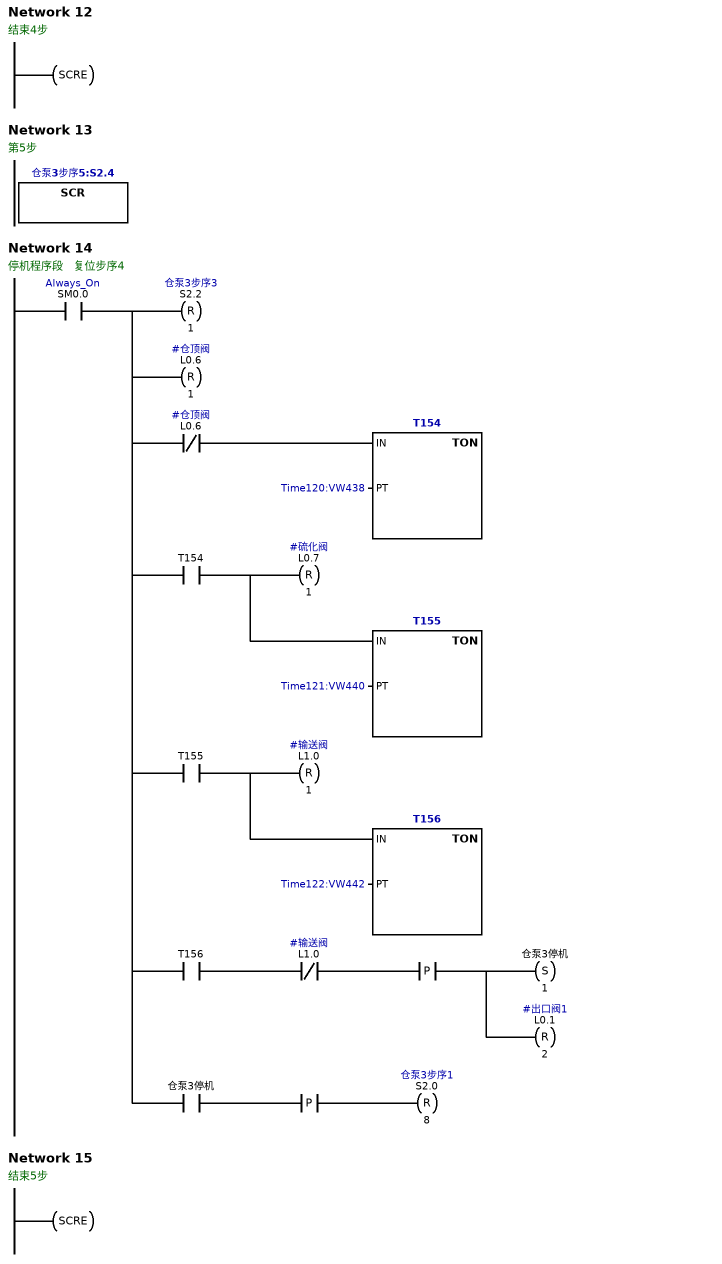
[picture p48: SBR18 networks 12-15]
Network 12
// 结束4步
SCRE
Network 13
// 第5步 
LSCR   仓泵3步序5:S2.4
Network 14
// 停机程序段   复位步序4 
// (network saved uncompiled; LAD cells follow)
// row 0: c0 -| |- Always_On:SM0.0 v  c1 -(R) 仓泵3步序3:S2.2, 1
// row 1: c0 ^v  c1 -(R) #仓顶阀:L0.6, 1
// row 2: c0 ^v  c1 -|/|- #仓顶阀:L0.6  c2 --  c3 [TON T154 IN:=power@row2, PT:=Time120:VW438]
// row 3: c0 ^v  c3 [box]
// row 4: c0 ^v  c1 -| |- T154 v  c2 -(R) #硫化阀:L0.7, 1
// row 5: c0 ^v  c1 ^  c2 --  c3 [TON T155 IN:=power@row5, PT:=Time121:VW440]
// row 6: c0 ^v  c3 [box]
// row 7: c0 ^v  c1 -| |- T155 v  c2 -(R) #输送阀:L1.0, 1
// row 8: c0 ^v  c1 ^  c2 --  c3 [TON T156 IN:=power@row8, PT:=Time122:VW442]
// row 9: c0 ^v  c3 [box]
// row 10: c0 ^v  c1 -| |- T156  c2 -|/|- #输送阀:L1.0  c3 -|P|-  v  c4 -(S) 仓泵3停机, 1
// row 11: c0 ^v  c3 ^  c4 -(R) #出口阀1:L0.1, 2
// row 12: c0 ^  c1 -| |- 仓泵3停机  c2 -|P|-  c3 -(R) 仓泵3步序1:S2.0, 8
Network 15
// 结束5步
SCRE
END_SUBROUTINE_BLOCK

SUBROUTINE_BLOCK 除尘器下料1:SBR19
TITLE=除尘器下料程序子程序说明   ：该子程序可用于除尘器下料程序  调用该子程序只需要填好子程序接口参数   然后核对子程序内部计数器有没有重复使用  有重复更改计数器  没有重复填好接口参数可直接使用
// 
// 从上往下依次的子程序接口
// 
// 使能
//  除尘器下料许可
// 系统错误
// 除尘器下料上下阀门自动位
// 除尘器下料阀上部Q点
// 除尘器下料阀下部Q点
// 除尘器气锤自动位
// 除尘器气碟自动位
// 除尘器中转气锤自动位
// 除尘器中转气碟自动位
// 上部阀门设定次数
// 下部阀门设定次数
// 上部阀门显示次数
// 下部阀门显示次数
VAR_INPUT
Sure:BOOL;	// L0.0 除尘器下料许可
END_VAR
VAR_IN_OUT
Error:BOOL;	// L0.1 系统错误
除尘器下料阀:BOOL;	// L0.2 除尘器下料阀ZD位 驱动两个阀门上下交替运行
除尘器下料阀上部:BOOL;	// L0.3 下料阀的上部阀门
除尘器下料阀下部:BOOL;	// L0.4 下料阀的下部阀门
除尘器气锤:BOOL;	// L0.5 气锤
除尘器气碟:BOOL;	// L0.6 气碟
除尘器中转气锤:BOOL;	// L0.7 中转气锤
除尘器中转气碟:BOOL;	// L1.0 中转气碟
上部次数设定:INT;	// LW2 上部阀运行次数设定
下部次数设定:INT;	// LW4 下部阀运行次数设定
上部次数显示:INT;	// LW6 上部阀运行次数显示
下部次数显示:INT;	// LW8 下部阀运行次数显示
END_VAR
BEGIN
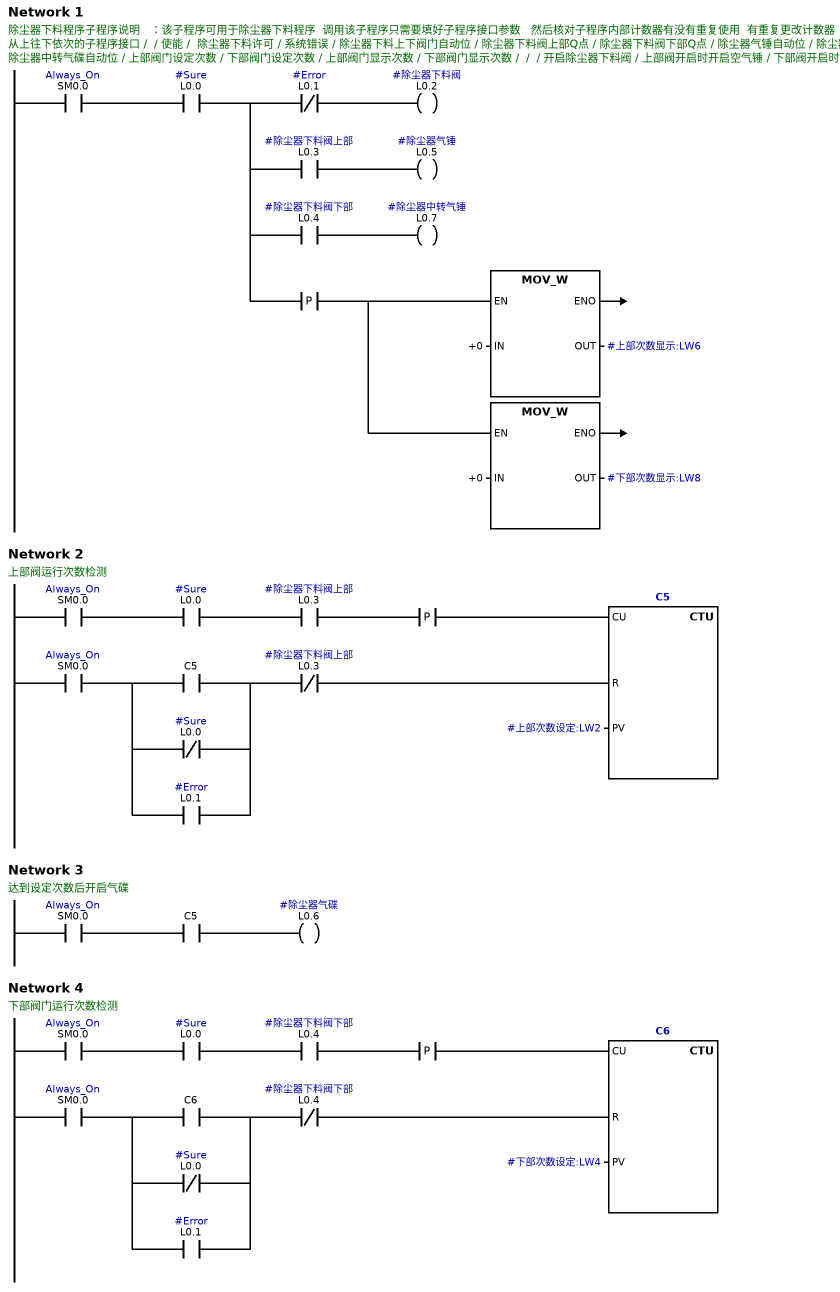
Network 1
// 除尘器下料程序子程序说明   ：该子程序可用于除尘器下料程序  调用该子程序只需要填好子程序接口参数   然后核对子程序内部计数器有没有重复使用  有重复更改计数器  没有重复填好接口参数可直接使用
// 
// 从上往下依次的子程序接口
// 
// 使能
//  除尘器下料许可
// 系统错误
// 除尘器下料上下阀门自动位
// 除尘器下料阀上部Q点
// 除尘器下料阀下部Q点
// 除尘器气锤自动位
// 除尘器气碟自动位
// 除尘器中转气锤自动位
// 除尘器中转气碟自动位
// 上部阀门设定次数
// 下部阀门设定次数
// 上部阀门显示次数
// 下部阀门显示次数
// 
// 
// 开启除尘器下料阀
// 上部阀开启时开启空气锤
// 下部阀开启时开启中转空气锤1
// 上部阀开启设定次数后开启气碟
// 下部阀开启设定次数后开启中转
LD     Always_On:SM0.0
A      #Sure:L0.0
LPS
AN     #Error:L0.1
=      #除尘器下料阀:L0.2
LRD
A      #除尘器下料阀上部:L0.3
=      #除尘器气锤:L0.5
LRD
A      #除尘器下料阀下部:L0.4
=      #除尘器中转气锤:L0.7
LPP
EU
MOVW   +0, #上部次数显示:LW6
MOVW   +0, #下部次数显示:LW8
Network 2
// 上部阀运行次数检测
LD     Always_On:SM0.0
A      #Sure:L0.0
A      #除尘器下料阀上部:L0.3
EU
LD     Always_On:SM0.0
LD     C5
ON     #Sure:L0.0
O      #Error:L0.1
ALD
AN     #除尘器下料阀上部:L0.3
CTU    C5, #上部次数设定:LW2
Network 3
// 达到设定次数后开启气碟
LD     Always_On:SM0.0
A      C5
=      #除尘器气碟:L0.6
Network 4
// 下部阀门运行次数检测
LD     Always_On:SM0.0
A      #Sure:L0.0
A      #除尘器下料阀下部:L0.4
EU
LD     Always_On:SM0.0
LD     C6
ON     #Sure:L0.0
O      #Error:L0.1
ALD
AN     #除尘器下料阀下部:L0.4
CTU    C6, #下部次数设定:LW4
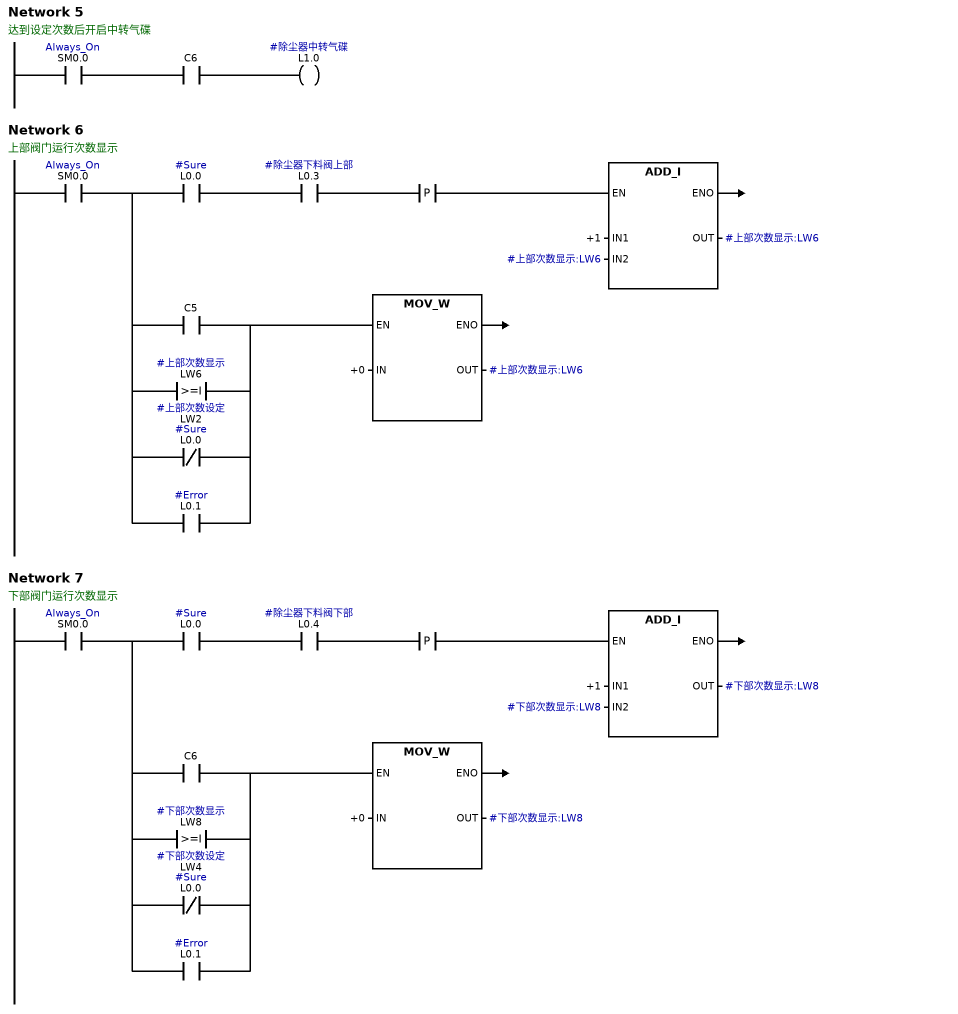
Network 5
// 达到设定次数后开启中转气碟
LD     Always_On:SM0.0
A      C6
=      #除尘器中转气碟:L1.0
Network 6
// 上部阀门运行次数显示
LD     Always_On:SM0.0
LPS
A      #Sure:L0.0
A      #除尘器下料阀上部:L0.3
EU
+I     +1, #上部次数显示:LW6
LPP
LD     C5
OW>=   #上部次数显示:LW6, #上部次数设定:LW2
ON     #Sure:L0.0
O      #Error:L0.1
ALD
MOVW   +0, #上部次数显示:LW6
Network 7
// 下部阀门运行次数显示
LD     Always_On:SM0.0
LPS
A      #Sure:L0.0
A      #除尘器下料阀下部:L0.4
EU
+I     +1, #下部次数显示:LW8
LPP
LD     C6
OW>=   #下部次数显示:LW8, #下部次数设定:LW4
ON     #Sure:L0.0
O      #Error:L0.1
ALD
MOVW   +0, #下部次数显示:LW8
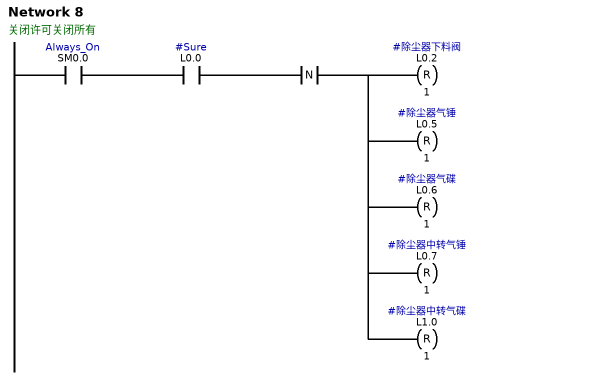
Network 8
// 关闭许可关闭所有
LD     Always_On:SM0.0
A      #Sure:L0.0
ED
R      #除尘器下料阀:L0.2, 1
R      #除尘器气锤:L0.5, 1
R      #除尘器气碟:L0.6, 1
R      #除尘器中转气锤:L0.7, 1
R      #除尘器中转气碟:L1.0, 1
END_SUBROUTINE_BLOCK

SUBROUTINE_BLOCK PauseUpValve5Group:SBR20
TITLE=
VAR_IN_OUT
Hand:BOOL;	// L0.0 手动信号
Auto:BOOL;	// L0.1 自动信号
Err:BOOL;	// L0.2 系统故障
UpValve1:BOOL;	// L0.3 提升阀1
UpValve2:BOOL;	// L0.4 提升阀2
UpValve3:BOOL;	// L0.5 提升阀3
UpValve4:BOOL;	// L0.6 提升阀4
UpValve5:BOOL;	// L0.7 提升阀5
Pulse1:BOOL;	// L1.0 脉冲阀1
Pulse2:BOOL;	// L1.1 脉冲阀2
Pulse3:BOOL;	// L1.2 脉冲阀3
Pulse4:BOOL;	// L1.3 脉冲阀4
Pulse5:BOOL;	// L1.4 脉冲阀5
UpValveRuntime:INT;	// LW2 提举阀运行时间
UpValveStoptime:INT;	// LW4 提举阀停止时间
PulseRuntime:INT;	// LW6 脉冲阀运行时间
PulseStoptime:INT;	// LW8 脉冲阀停止时间
END_VAR
BEGIN
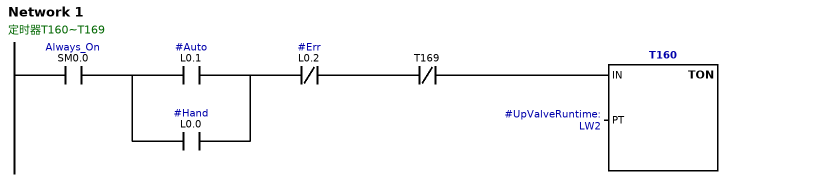
Network 1
// 定时器T160~T169
LD     Always_On:SM0.0
LD     #Auto:L0.1
O      #Hand:L0.0
ALD
AN     #Err:L0.2
AN     T169
TON    T160, #UpValveRuntime:LW2
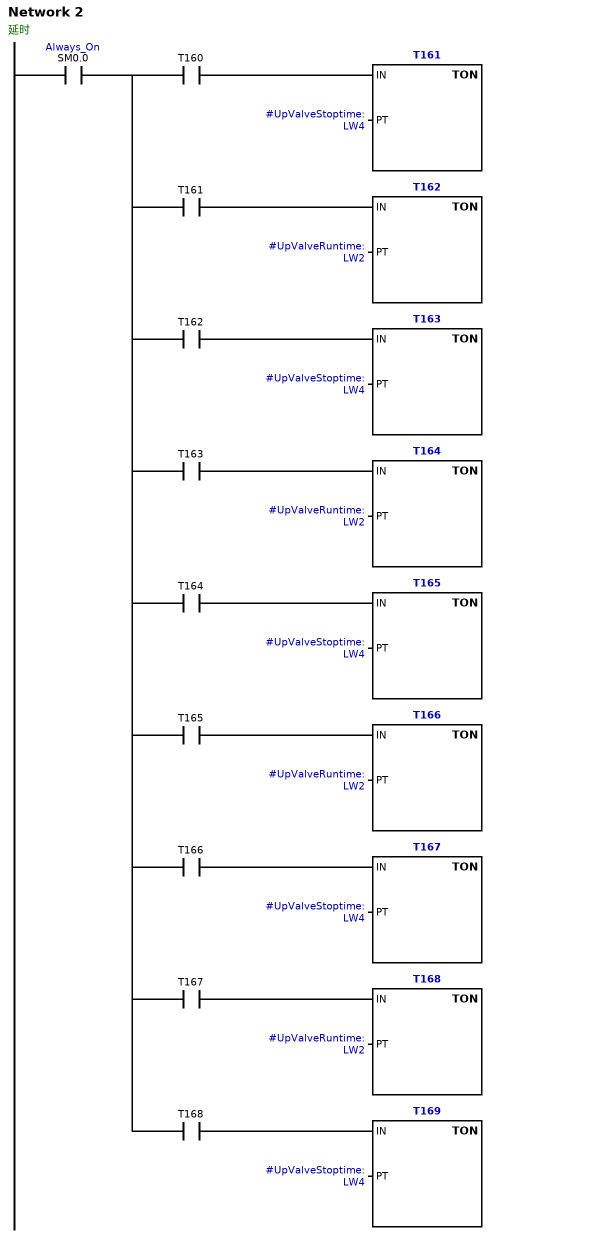
Network 2
// 延时
LD     Always_On:SM0.0
LPS
A      T160
TON    T161, #UpValveStoptime:LW4
LRD
A      T161
TON    T162, #UpValveRuntime:LW2
LRD
A      T162
TON    T163, #UpValveStoptime:LW4
LRD
A      T163
TON    T164, #UpValveRuntime:LW2
LRD
A      T164
TON    T165, #UpValveStoptime:LW4
LRD
A      T165
TON    T166, #UpValveRuntime:LW2
LRD
A      T166
TON    T167, #UpValveStoptime:LW4
LRD
A      T167
TON    T168, #UpValveRuntime:LW2
LPP
A      T168
TON    T169, #UpValveStoptime:LW4
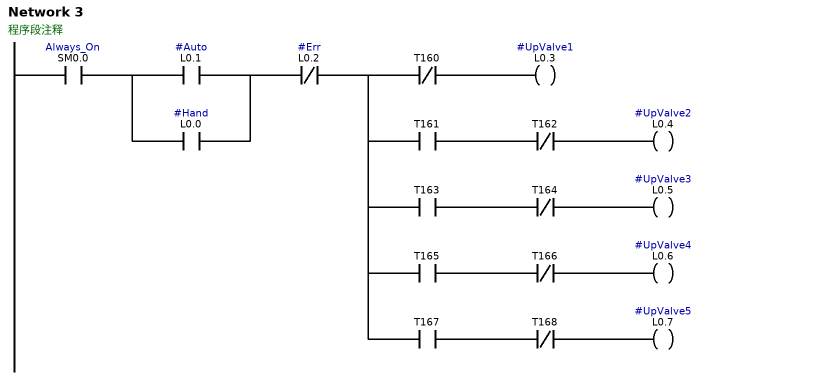
Network 3
//  程序段注释
LD     Always_On:SM0.0
LD     #Auto:L0.1
O      #Hand:L0.0
ALD
AN     #Err:L0.2
LPS
AN     T160
=      #UpValve1:L0.3
LRD
A      T161
AN     T162
=      #UpValve2:L0.4
LRD
A      T163
AN     T164
=      #UpValve3:L0.5
LRD
A      T165
AN     T166
=      #UpValve4:L0.6
LPP
A      T167
AN     T168
=      #UpValve5:L0.7
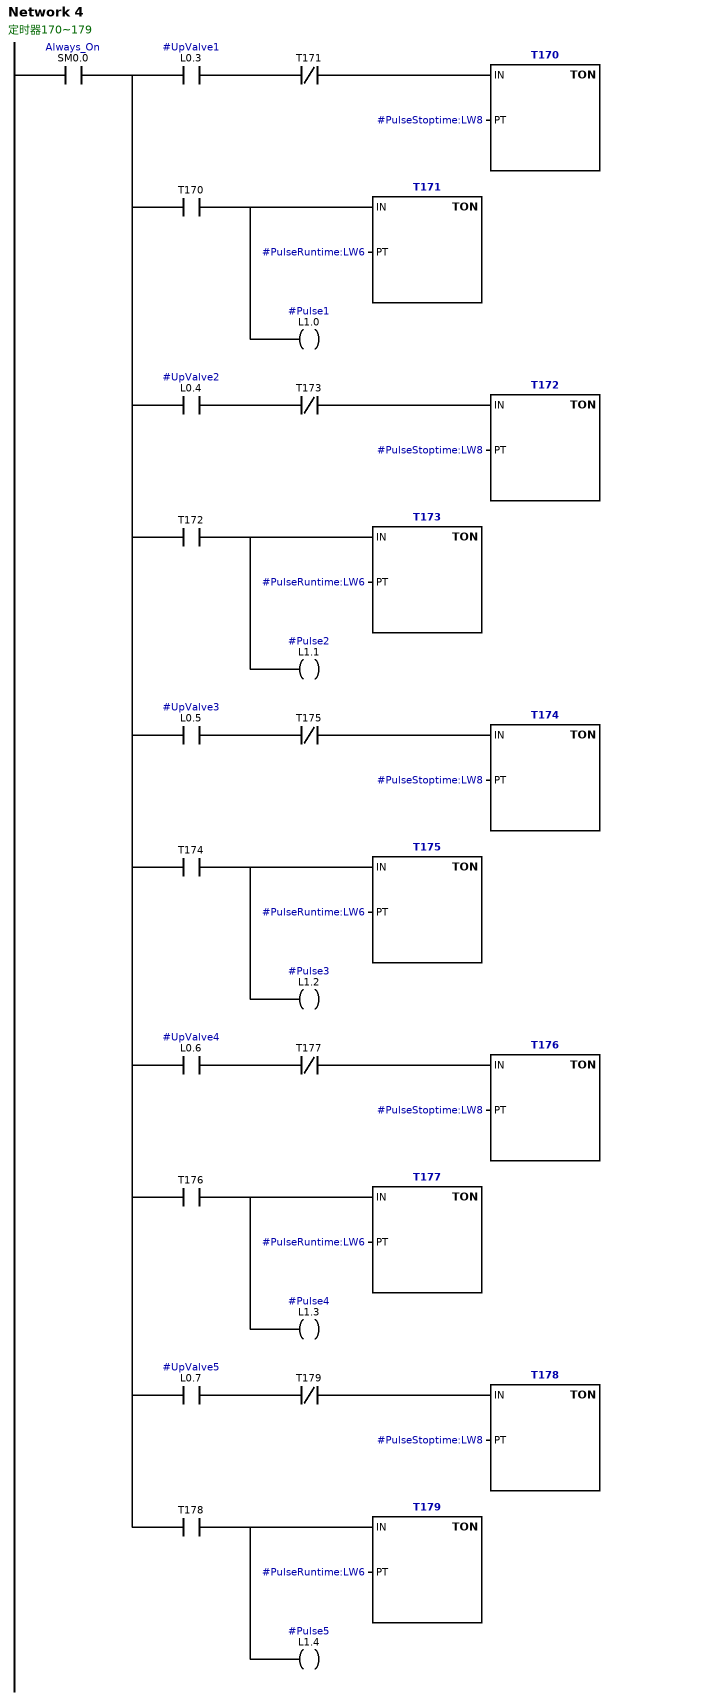
Network 4
// 定时器170~179
LD     Always_On:SM0.0
LPS
A      #UpValve1:L0.3
AN     T171
TON    T170, #PulseStoptime:LW8
LRD
A      T170
TON    T171, #PulseRuntime:LW6
=      #Pulse1:L1.0
LRD
A      #UpValve2:L0.4
AN     T173
TON    T172, #PulseStoptime:LW8
LRD
A      T172
TON    T173, #PulseRuntime:LW6
=      #Pulse2:L1.1
LRD
A      #UpValve3:L0.5
AN     T175
TON    T174, #PulseStoptime:LW8
LRD
A      T174
TON    T175, #PulseRuntime:LW6
=      #Pulse3:L1.2
LRD
A      #UpValve4:L0.6
AN     T177
TON    T176, #PulseStoptime:LW8
LRD
A      T176
TON    T177, #PulseRuntime:LW6
=      #Pulse4:L1.3
LRD
A      #UpValve5:L0.7
AN     T179
TON    T178, #PulseStoptime:LW8
LPP
A      T178
TON    T179, #PulseRuntime:LW6
=      #Pulse5:L1.4
END_SUBROUTINE_BLOCK

SUBROUTINE_BLOCK 双除尘器切换1:SBR21
TITLE=
VAR_INPUT
IN_T1:BOOL;	// L0.0 
IN_T2:BOOL;	// L0.1 
END_VAR
VAR_IN_OUT
进口阀1:BOOL;	// L0.2 
出口阀1:BOOL;	// L0.3 
脉冲仪1:BOOL;	// L0.4 
进口阀2:BOOL;	// L0.5 
出口阀2:BOOL;	// L0.6 
脉冲仪2:BOOL;	// L0.7 
引风机1:BOOL;	// L1.0 
引风机2:BOOL;	// L1.1 
State1:BOOL;	// L1.2 除尘器1 切换中
State2:BOOL;	// L1.3 除尘器2 切换中
END_VAR
BEGIN
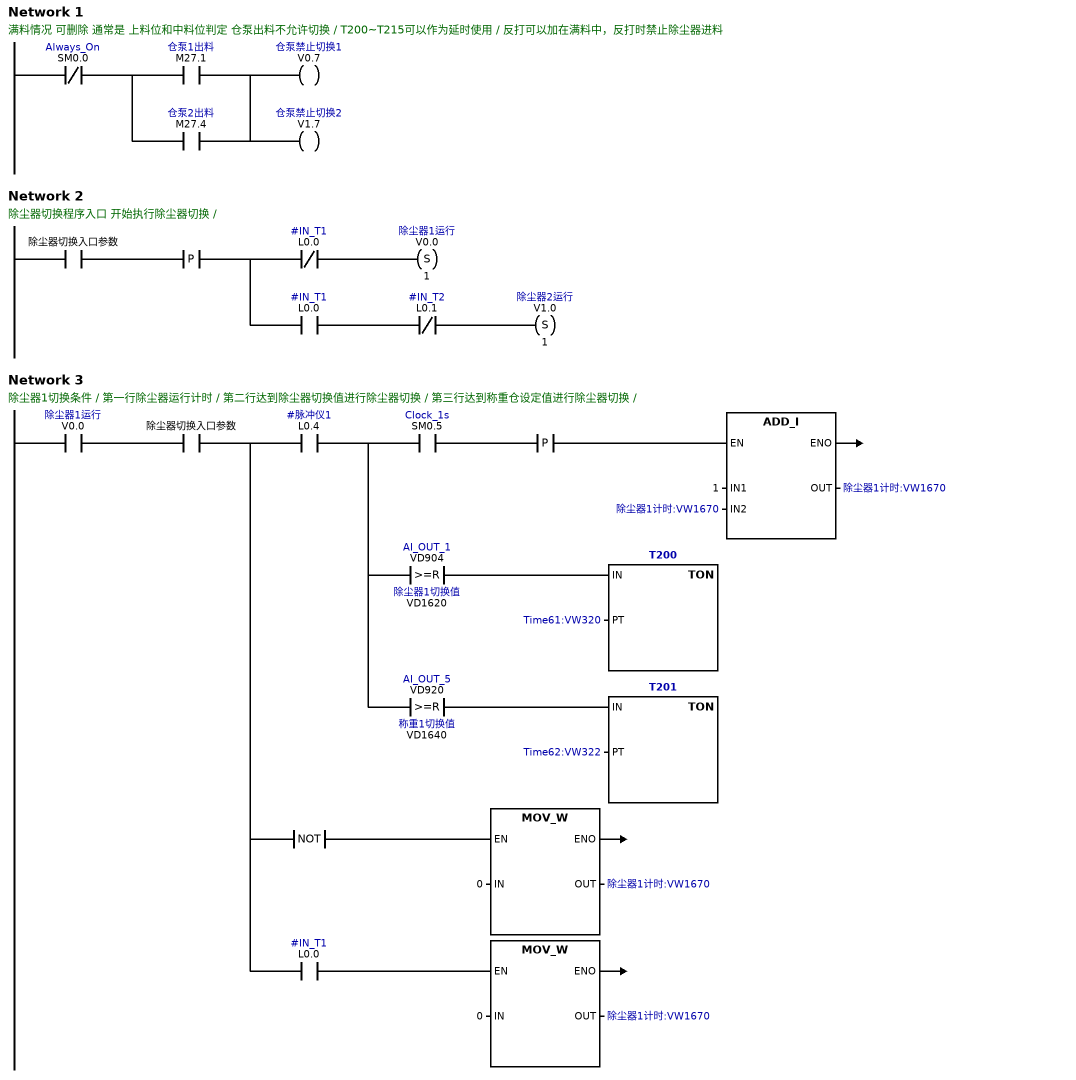
Network 1
// 满料情况 可删除 通常是 上料位和中料位判定 仓泵出料不允许切换
// T200~T215可以作为延时使用
// 反打可以加在满料中，反打时禁止除尘器进料
LDN    Always_On:SM0.0
LD     仓泵1出料:M27.1
O      仓泵2出料:M27.4
ALD
=      仓泵禁止切换1:V0.7
=      仓泵禁止切换2:V1.7
Network 2
//  除尘器切换程序入口 开始执行除尘器切换
// 
// (network saved uncompiled; LAD cells follow)
// row 0: c0 -| |- 除尘器切换入口参数  c1 -|P|-  v  c2 -|/|- #IN_T1:L0.0  c3 -(S) 除尘器1运行:V0.0, 1
// row 1: c1 ^  c2 -| |- #IN_T1:L0.0  c3 -|/|- #IN_T2:L0.1  c4 -(S) 除尘器2运行:V1.0, 1
Network 3
// 除尘器1切换条件
// 第一行除尘器运行计时
// 第二行达到除尘器切换值进行除尘器切换
// 第三行达到称重仓设定值进行除尘器切换
// 
// (network saved uncompiled; LAD cells follow)
// row 0: c0 -| |- 除尘器1运行:V0.0  c1 -| |- 除尘器切换入口参数 v  c2 -| |- #脉冲仪1:L0.4 v  c3 -| |- Clock_1s:SM0.5  c4 -|P|-  c5 --  c6 [ADD_I EN:=power@row0, IN1:=1, IN2:=除尘器1计时:VW1670, ENO=>power, OUT=>除尘器1计时:VW1670]  c7 ->
// row 1: c1 ^v  c2 ^v  c6 [box]
// row 2: c1 ^v  c2 ^v  c3 -|>=R|- AI_OUT_1:VD904, 除尘器1切换值:VD1620  c4 --  c5 [TON T200 IN:=power@row2, PT:=Time61:VW320]
// row 3: c1 ^v  c2 ^v  c5 [box]
// row 4: c1 ^v  c2 ^  c3 -|>=R|- AI_OUT_5:VD920, 称重1切换值:VD1640  c4 --  c5 [TON T201 IN:=power@row4, PT:=Time62:VW322]
// row 5: c1 ^v  c5 [box]
// row 6: c1 ^v  c2 -|NOT|-  c3 --  c4 [MOV_W EN:=power@row6, IN:=0, ENO=>power, OUT=>除尘器1计时:VW1670]  c5 ->
// row 7: c1 ^v  c4 [box]
// row 8: c1 ^  c2 -| |- #IN_T1:L0.0  c3 --  c4 [MOV_W EN:=power@row8, IN:=0, ENO=>power, OUT=>除尘器1计时:VW1670]  c5 ->
// row 9: c4 [box]
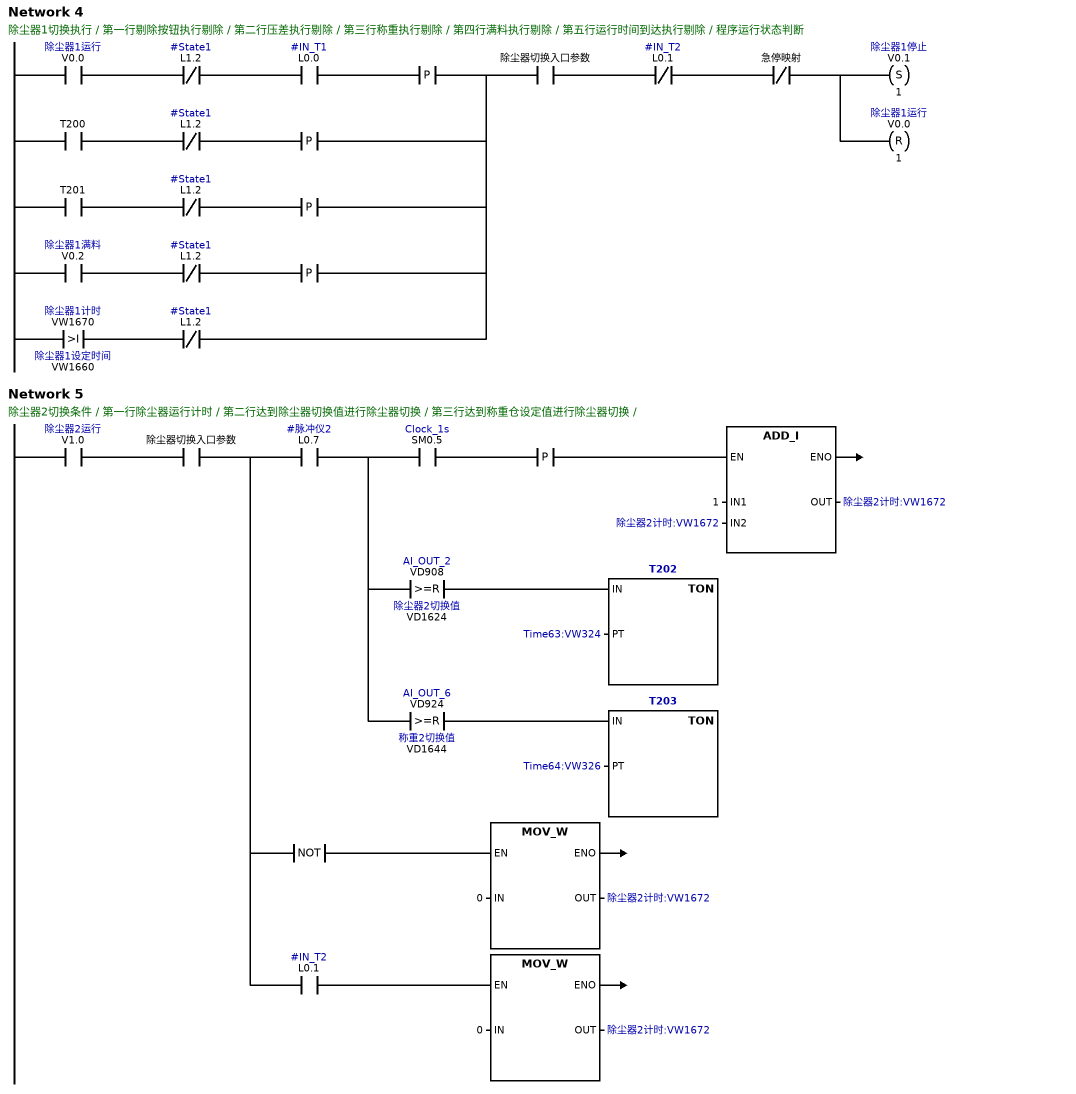
Network 4
// 除尘器1切换执行
// 第一行剔除按钮执行剔除
// 第二行压差执行剔除
// 第三行称重执行剔除
// 第四行满料执行剔除
// 第五行运行时间到达执行剔除
// 程序运行状态判断
// (network saved uncompiled; LAD cells follow)
// row 0: c0 -| |- 除尘器1运行:V0.0  c1 -|/|- #State1:L1.2  c2 -| |- #IN_T1:L0.0  c3 -|P|-  v  c4 -| |- 除尘器切换入口参数  c5 -|/|- #IN_T2:L0.1  c6 -|/|- 急停映射 v  c7 -(S) 除尘器1停止:V0.1, 1
// row 1: c0 -| |- T200  c1 -|/|- #State1:L1.2  c2 -|P|-  c3 -- ^v  c6 ^  c7 -(R) 除尘器1运行:V0.0, 1
// row 2: c0 -| |- T201  c1 -|/|- #State1:L1.2  c2 -|P|-  c3 -- ^v
// row 3: c0 -| |- 除尘器1满料:V0.2  c1 -|/|- #State1:L1.2  c2 -|P|-  c3 -- ^v
// row 4: c0 -|>I|- 除尘器1计时:VW1670, 除尘器1设定时间:VW1660  c1 -|/|- #State1:L1.2  c2 --  c3 -- ^
Network 5
// 除尘器2切换条件
// 第一行除尘器运行计时
// 第二行达到除尘器切换值进行除尘器切换
// 第三行达到称重仓设定值进行除尘器切换
// 
// (network saved uncompiled; LAD cells follow)
// row 0: c0 -| |- 除尘器2运行:V1.0  c1 -| |- 除尘器切换入口参数 v  c2 -| |- #脉冲仪2:L0.7 v  c3 -| |- Clock_1s:SM0.5  c4 -|P|-  c5 --  c6 [ADD_I EN:=power@row0, IN1:=1, IN2:=除尘器2计时:VW1672, ENO=>power, OUT=>除尘器2计时:VW1672]  c7 ->
// row 1: c1 ^v  c2 ^v  c6 [box]
// row 2: c1 ^v  c2 ^v  c3 -|>=R|- AI_OUT_2:VD908, 除尘器2切换值:VD1624  c4 --  c5 [TON T202 IN:=power@row2, PT:=Time63:VW324]
// row 3: c1 ^v  c2 ^v  c5 [box]
// row 4: c1 ^v  c2 ^  c3 -|>=R|- AI_OUT_6:VD924, 称重2切换值:VD1644  c4 --  c5 [TON T203 IN:=power@row4, PT:=Time64:VW326]
// row 5: c1 ^v  c5 [box]
// row 6: c1 ^v  c2 -|NOT|-  c3 --  c4 [MOV_W EN:=power@row6, IN:=0, ENO=>power, OUT=>除尘器2计时:VW1672]  c5 ->
// row 7: c1 ^v  c4 [box]
// row 8: c1 ^  c2 -| |- #IN_T2:L0.1  c3 --  c4 [MOV_W EN:=power@row8, IN:=0, ENO=>power, OUT=>除尘器2计时:VW1672]  c5 ->
// row 9: c4 [box]
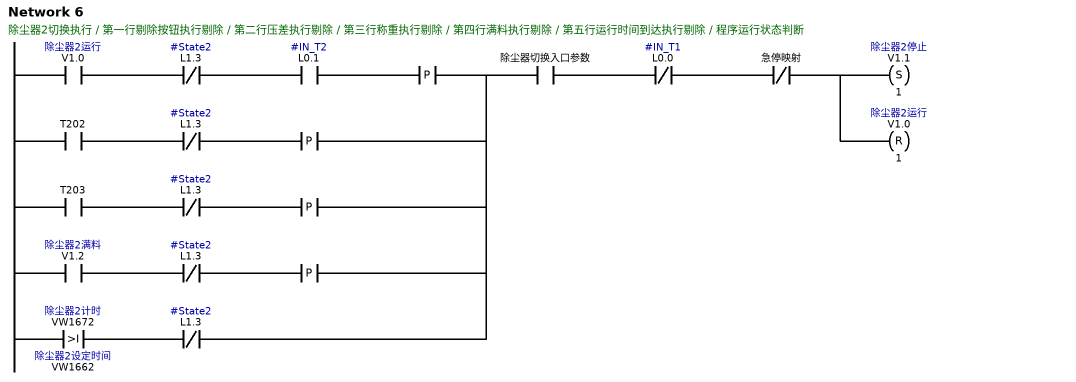
Network 6
// 除尘器2切换执行
// 第一行剔除按钮执行剔除
// 第二行压差执行剔除
// 第三行称重执行剔除
// 第四行满料执行剔除
// 第五行运行时间到达执行剔除
// 程序运行状态判断
// (network saved uncompiled; LAD cells follow)
// row 0: c0 -| |- 除尘器2运行:V1.0  c1 -|/|- #State2:L1.3  c2 -| |- #IN_T2:L0.1  c3 -|P|-  v  c4 -| |- 除尘器切换入口参数  c5 -|/|- #IN_T1:L0.0  c6 -|/|- 急停映射 v  c7 -(S) 除尘器2停止:V1.1, 1
// row 1: c0 -| |- T202  c1 -|/|- #State2:L1.3  c2 -|P|-  c3 -- ^v  c6 ^  c7 -(R) 除尘器2运行:V1.0, 1
// row 2: c0 -| |- T203  c1 -|/|- #State2:L1.3  c2 -|P|-  c3 -- ^v
// row 3: c0 -| |- 除尘器2满料:V1.2  c1 -|/|- #State2:L1.3  c2 -|P|-  c3 -- ^v
// row 4: c0 -|>I|- 除尘器2计时:VW1672, 除尘器2设定时间:VW1662  c1 -|/|- #State2:L1.3  c2 --  c3 -- ^
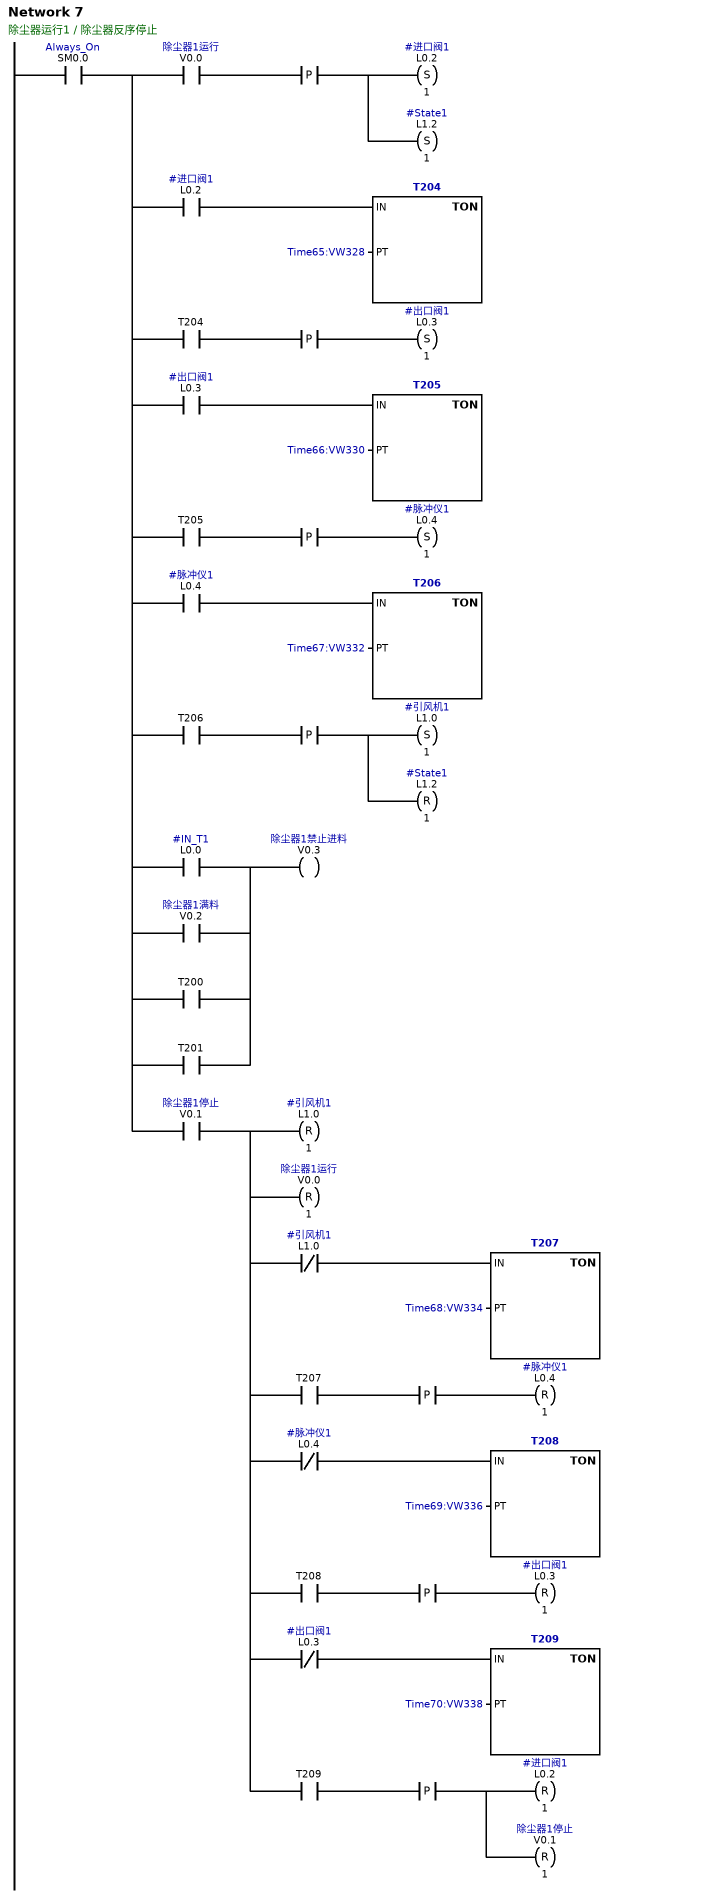
Network 7
// 除尘器运行1
// 除尘器反序停止
LD     Always_On:SM0.0
LPS
A      除尘器1运行:V0.0
EU
S      #进口阀1:L0.2, 1
S      #State1:L1.2, 1
LRD
LPS
A      #进口阀1:L0.2
TON    T204, Time65:VW328
LRD
A      T204
EU
S      #出口阀1:L0.3, 1
LRD
A      #出口阀1:L0.3
TON    T205, Time66:VW330
LRD
A      T205
EU
S      #脉冲仪1:L0.4, 1
LPP
A      #脉冲仪1:L0.4
TON    T206, Time67:VW332
LRD
A      T206
EU
S      #引风机1:L1.0, 1
R      #State1:L1.2, 1
LRD
LD     #IN_T1:L0.0
O      除尘器1满料:V0.2
O      T200
O      T201
ALD
=      除尘器1禁止进料:V0.3
LPP
A      除尘器1停止:V0.1
LPS
R      #引风机1:L1.0, 1
R      除尘器1运行:V0.0, 1
AN     #引风机1:L1.0
TON    T207, Time68:VW334
LRD
A      T207
EU
R      #脉冲仪1:L0.4, 1
LRD
AN     #脉冲仪1:L0.4
TON    T208, Time69:VW336
LRD
A      T208
EU
R      #出口阀1:L0.3, 1
LRD
AN     #出口阀1:L0.3
TON    T209, Time70:VW338
LPP
A      T209
EU
R      #进口阀1:L0.2, 1
R      除尘器1停止:V0.1, 1
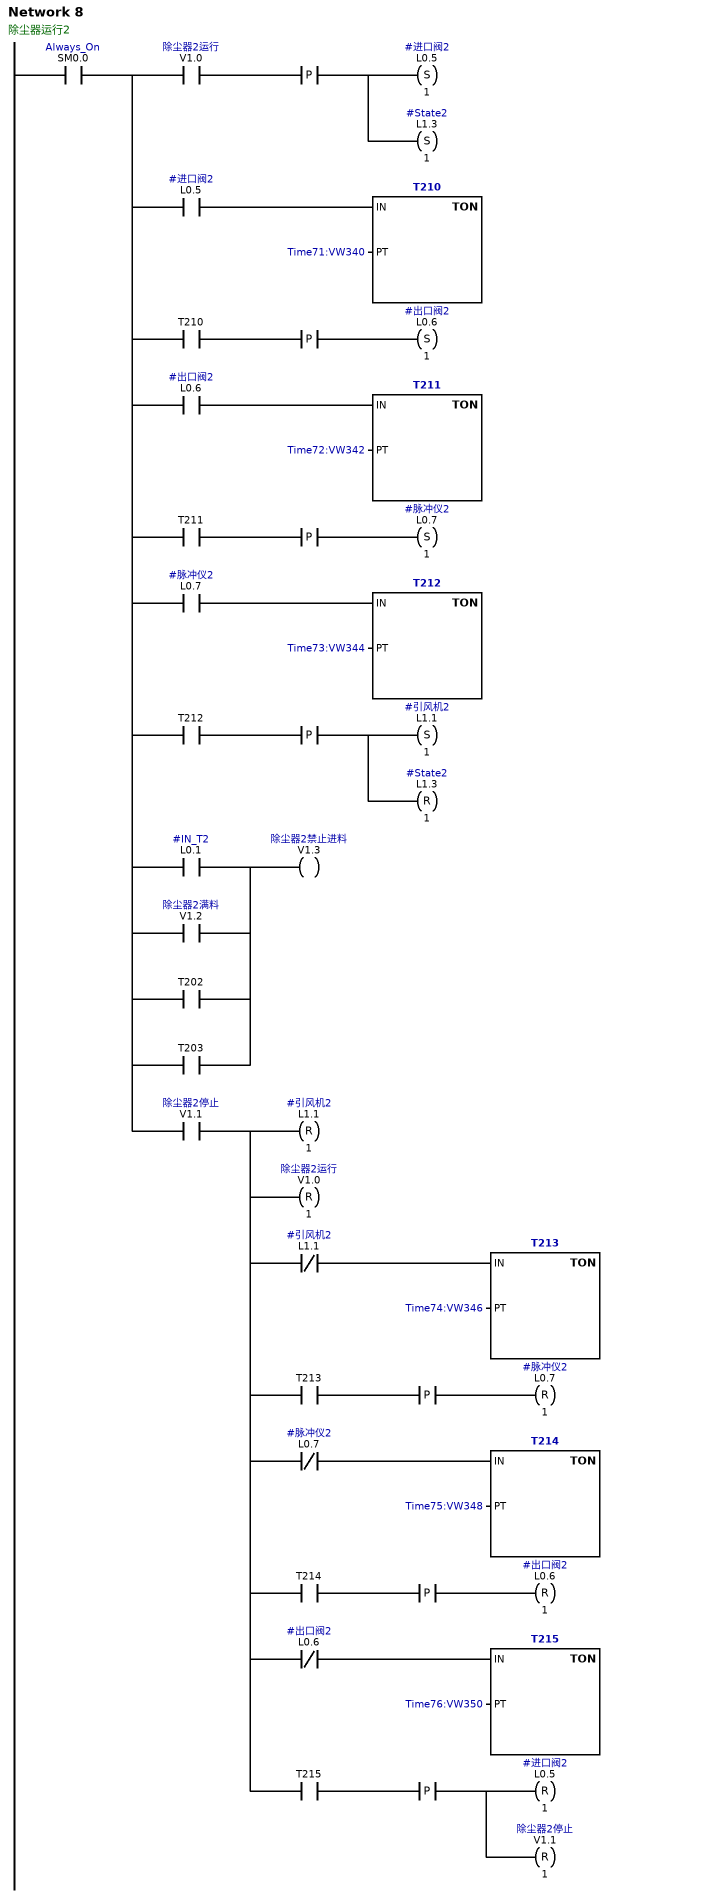
Network 8
// 除尘器运行2
LD     Always_On:SM0.0
LPS
A      除尘器2运行:V1.0
EU
S      #进口阀2:L0.5, 1
S      #State2:L1.3, 1
LRD
LPS
A      #进口阀2:L0.5
TON    T210, Time71:VW340
LRD
A      T210
EU
S      #出口阀2:L0.6, 1
LRD
A      #出口阀2:L0.6
TON    T211, Time72:VW342
LRD
A      T211
EU
S      #脉冲仪2:L0.7, 1
LPP
A      #脉冲仪2:L0.7
TON    T212, Time73:VW344
LRD
A      T212
EU
S      #引风机2:L1.1, 1
R      #State2:L1.3, 1
LRD
LD     #IN_T2:L0.1
O      除尘器2满料:V1.2
O      T202
O      T203
ALD
=      除尘器2禁止进料:V1.3
LPP
A      除尘器2停止:V1.1
LPS
R      #引风机2:L1.1, 1
R      除尘器2运行:V1.0, 1
AN     #引风机2:L1.1
TON    T213, Time74:VW346
LRD
A      T213
EU
R      #脉冲仪2:L0.7, 1
LRD
AN     #脉冲仪2:L0.7
TON    T214, Time75:VW348
LRD
A      T214
EU
R      #出口阀2:L0.6, 1
LRD
AN     #出口阀2:L0.6
TON    T215, Time76:VW350
LPP
A      T215
EU
R      #进口阀2:L0.5, 1
R      除尘器2停止:V1.1, 1
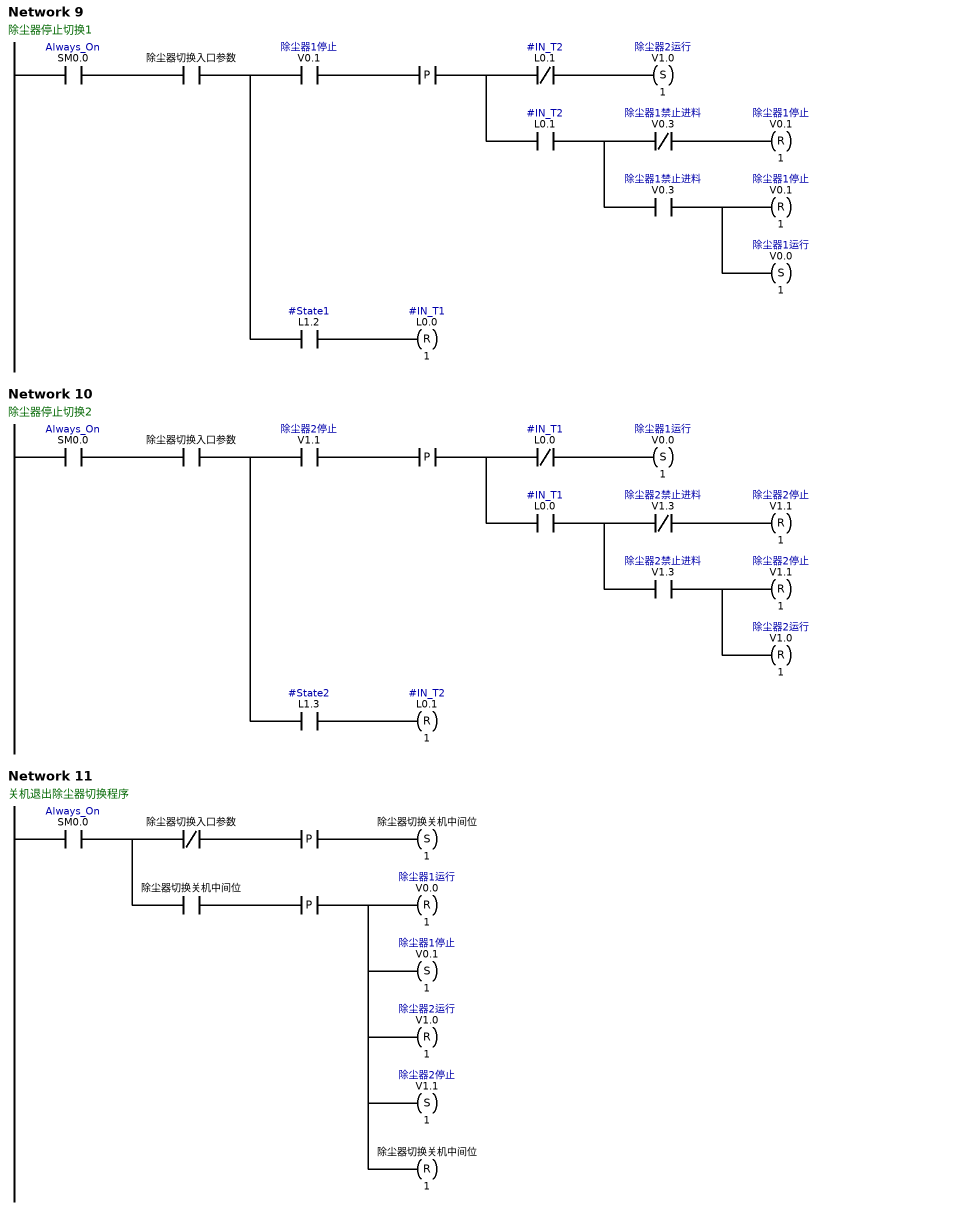
Network 9
// 除尘器停止切换1
// (network saved uncompiled; LAD cells follow)
// row 0: c0 -| |- Always_On:SM0.0  c1 -| |- 除尘器切换入口参数 v  c2 -| |- 除尘器1停止:V0.1  c3 -|P|-  v  c4 -|/|- #IN_T2:L0.1  c5 -(S) 除尘器2运行:V1.0, 1
// row 1: c1 ^v  c3 ^  c4 -| |- #IN_T2:L0.1 v  c5 -|/|- 除尘器1禁止进料:V0.3  c6 -(R) 除尘器1停止:V0.1, 1
// row 2: c1 ^v  c4 ^  c5 -| |- 除尘器1禁止进料:V0.3 v  c6 -(R) 除尘器1停止:V0.1, 1
// row 3: c1 ^v  c5 ^  c6 -(S) 除尘器1运行:V0.0, 1
// row 4: c1 ^  c2 -| |- #State1:L1.2  c3 -(R) #IN_T1:L0.0, 1
Network 10
// 除尘器停止切换2
// (network saved uncompiled; LAD cells follow)
// row 0: c0 -| |- Always_On:SM0.0  c1 -| |- 除尘器切换入口参数 v  c2 -| |- 除尘器2停止:V1.1  c3 -|P|-  v  c4 -|/|- #IN_T1:L0.0  c5 -(S) 除尘器1运行:V0.0, 1
// row 1: c1 ^v  c3 ^  c4 -| |- #IN_T1:L0.0 v  c5 -|/|- 除尘器2禁止进料:V1.3  c6 -(R) 除尘器2停止:V1.1, 1
// row 2: c1 ^v  c4 ^  c5 -| |- 除尘器2禁止进料:V1.3 v  c6 -(R) 除尘器2停止:V1.1, 1
// row 3: c1 ^v  c5 ^  c6 -(R) 除尘器2运行:V1.0, 1
// row 4: c1 ^  c2 -| |- #State2:L1.3  c3 -(R) #IN_T2:L0.1, 1
Network 11
// 关机退出除尘器切换程序
// (network saved uncompiled; LAD cells follow)
// row 0: c0 -| |- Always_On:SM0.0 v  c1 -|/|- 除尘器切换入口参数  c2 -|P|-  c3 -(S) 除尘器切换关机中间位, 1
// row 1: c0 ^  c1 -| |- 除尘器切换关机中间位  c2 -|P|-  v  c3 -(R) 除尘器1运行:V0.0, 1
// row 2: c2 ^v  c3 -(S) 除尘器1停止:V0.1, 1
// row 3: c2 ^v  c3 -(R) 除尘器2运行:V1.0, 1
// row 4: c2 ^v  c3 -(S) 除尘器2停止:V1.1, 1
// row 5: c2 ^  c3 -(R) 除尘器切换关机中间位, 1
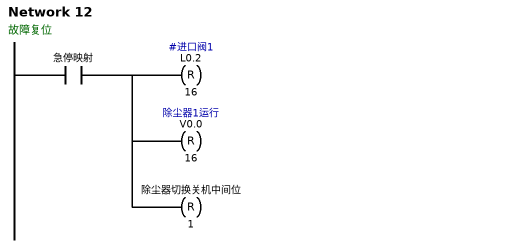
Network 12
// 故障复位
// (network saved uncompiled; LAD cells follow)
// row 0: c0 -| |- 急停映射 v  c1 -(R) #进口阀1:L0.2, 16
// row 1: c0 ^v  c1 -(R) 除尘器1运行:V0.0, 16
// row 2: c0 ^  c1 -(R) 除尘器切换关机中间位, 1
END_SUBROUTINE_BLOCK

SUBROUTINE_BLOCK PauseUpValve3Group:SBR22
TITLE=
VAR_IN_OUT
Hand:BOOL;	// L0.0 手动信号
Auto:BOOL;	// L0.1 自动信号
Err:BOOL;	// L0.2 系统故障
UpValve1:BOOL;	// L0.3 提升阀1
UpValve2:BOOL;	// L0.4 提升阀2
UpValve3:BOOL;	// L0.5 提升阀3
Pulse1:BOOL;	// L0.6 脉冲阀1
Pulse2:BOOL;	// L0.7 脉冲阀2
Pulse3:BOOL;	// L1.0 脉冲阀3
UpValveRuntime:INT;	// LW2 提举阀运行时间
UpValveStoptime:INT;	// LW4 提举阀停止时间
PulseRuntime:INT;	// LW6 脉冲阀运行时间
PulseStoptime:INT;	// LW8 脉冲阀停止时间
END_VAR
BEGIN
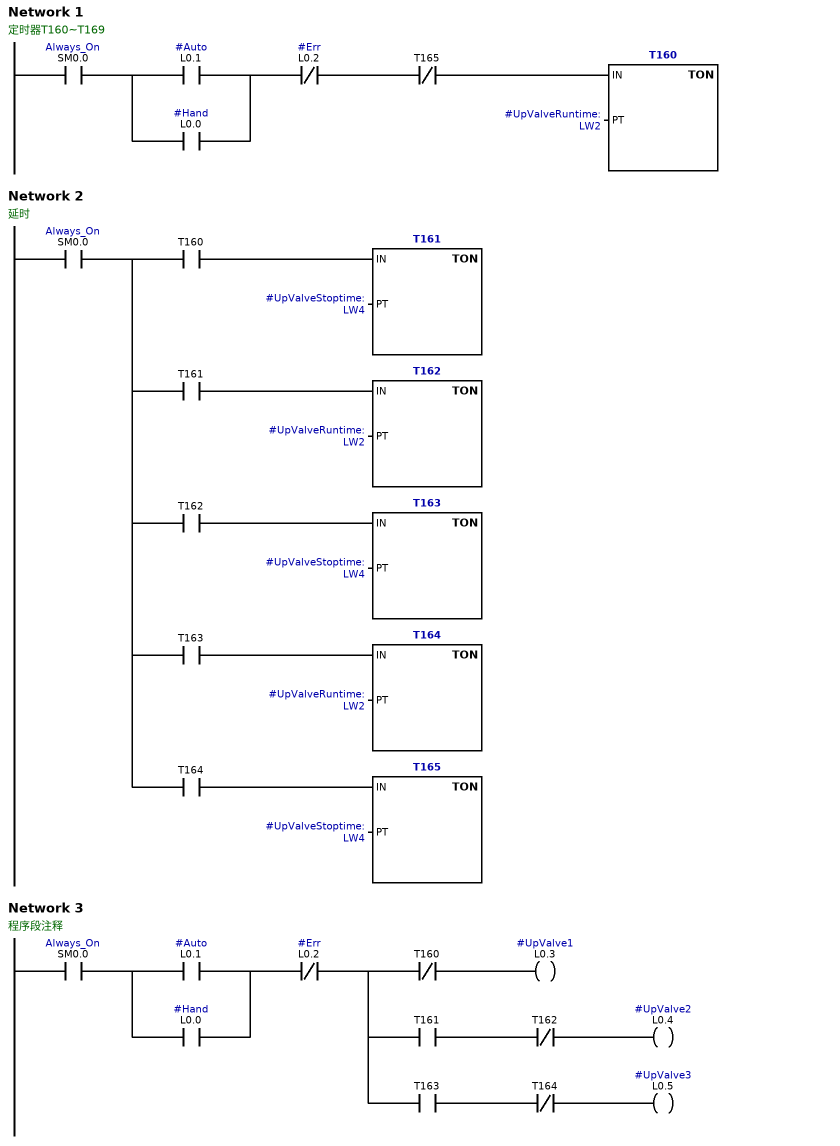
Network 1
// 定时器T160~T169
LD     Always_On:SM0.0
LD     #Auto:L0.1
O      #Hand:L0.0
ALD
AN     #Err:L0.2
AN     T165
TON    T160, #UpValveRuntime:LW2
Network 2
// 延时
LD     Always_On:SM0.0
LPS
A      T160
TON    T161, #UpValveStoptime:LW4
LRD
A      T161
TON    T162, #UpValveRuntime:LW2
LRD
A      T162
TON    T163, #UpValveStoptime:LW4
LRD
A      T163
TON    T164, #UpValveRuntime:LW2
LPP
A      T164
TON    T165, #UpValveStoptime:LW4
Network 3
//  程序段注释
LD     Always_On:SM0.0
LD     #Auto:L0.1
O      #Hand:L0.0
ALD
AN     #Err:L0.2
LPS
AN     T160
=      #UpValve1:L0.3
LRD
A      T161
AN     T162
=      #UpValve2:L0.4
LPP
A      T163
AN     T164
=      #UpValve3:L0.5
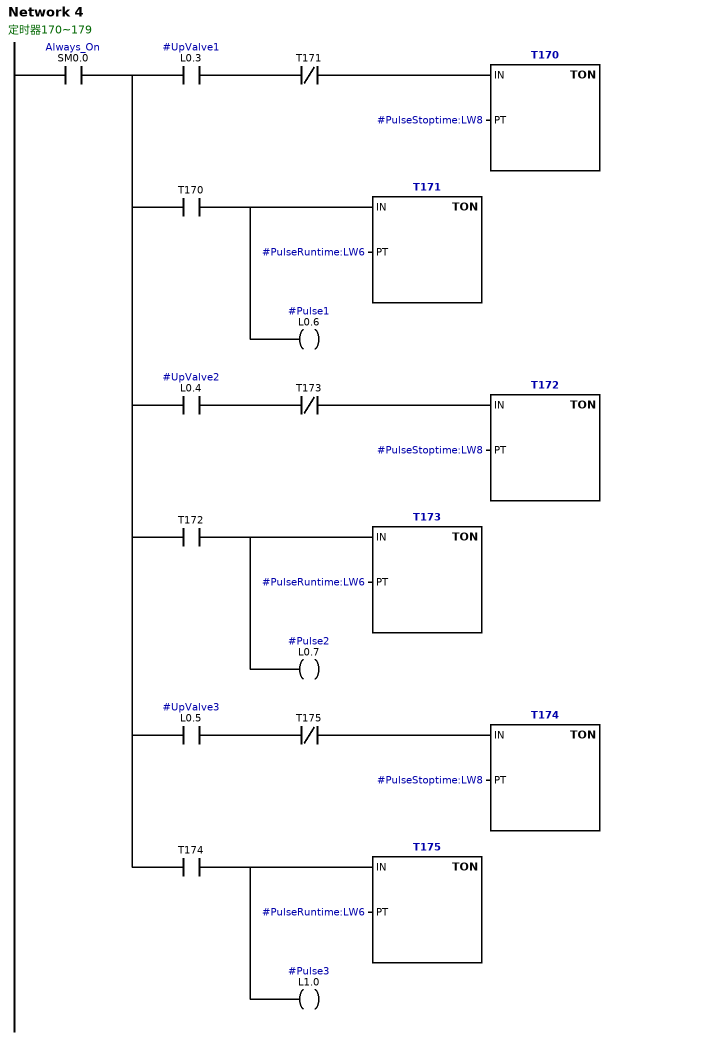
Network 4
// 定时器170~179
LD     Always_On:SM0.0
LPS
A      #UpValve1:L0.3
AN     T171
TON    T170, #PulseStoptime:LW8
LRD
A      T170
TON    T171, #PulseRuntime:LW6
=      #Pulse1:L0.6
LRD
A      #UpValve2:L0.4
AN     T173
TON    T172, #PulseStoptime:LW8
LRD
A      T172
TON    T173, #PulseRuntime:LW6
=      #Pulse2:L0.7
LRD
A      #UpValve3:L0.5
AN     T175
TON    T174, #PulseStoptime:LW8
LPP
A      T174
TON    T175, #PulseRuntime:LW6
=      #Pulse3:L1.0
END_SUBROUTINE_BLOCK

SUBROUTINE_BLOCK 仓泵4:SBR23
TITLE=
VAR_OUTPUT
出口阀:BOOL;	// L0.0 
呼吸阀:BOOL;	// L0.1 
进料阀:BOOL;	// L0.2 
进料阀上:BOOL;	// L0.3 
仓顶阀:BOOL;	// L0.4 
流化阀:BOOL;	// L0.5 
输送阀:BOOL;	// L0.6 
END_VAR
BEGIN
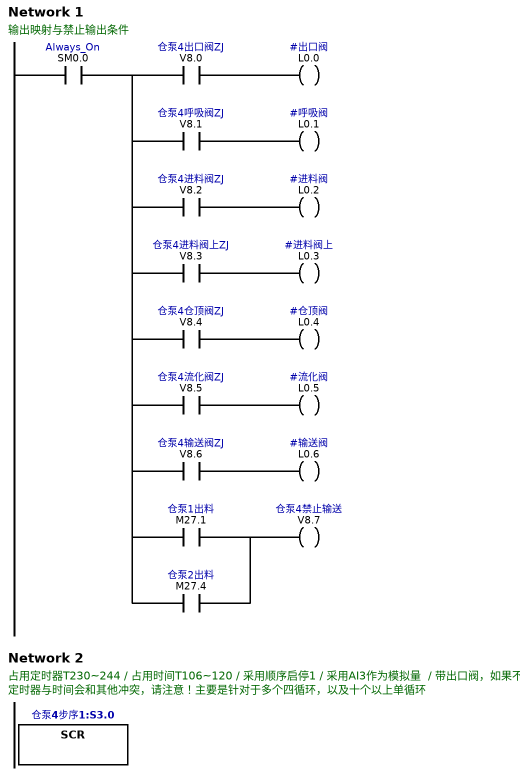
Network 1
// 输出映射与禁止输出条件
LD     Always_On:SM0.0
LPS
A      仓泵4出口阀ZJ:V8.0
=      #出口阀:L0.0
LRD
A      仓泵4呼吸阀ZJ:V8.1
=      #呼吸阀:L0.1
LRD
A      仓泵4进料阀ZJ:V8.2
=      #进料阀:L0.2
LRD
A      仓泵4进料阀上ZJ:V8.3
=      #进料阀上:L0.3
LRD
A      仓泵4仓顶阀ZJ:V8.4
=      #仓顶阀:L0.4
LRD
A      仓泵4流化阀ZJ:V8.5
=      #流化阀:L0.5
LRD
A      仓泵4输送阀ZJ:V8.6
=      #输送阀:L0.6
LPP
LD     仓泵1出料:M27.1
O      仓泵2出料:M27.4
ALD
=      仓泵4禁止输送:V8.7
Network 2
// 占用定时器T230~244
// 占用时间T106~120
// 采用顺序启停1
// 采用AI3作为模拟量 
// 带出口阀，如果不需要可删除
// 同时仅一个仓泵出料，多需求请改网络5
// 定时器与时间会和其他冲突，请注意！主要是针对于多个四循环，以及十个以上单循环
LSCR   仓泵4步序1:S3.0
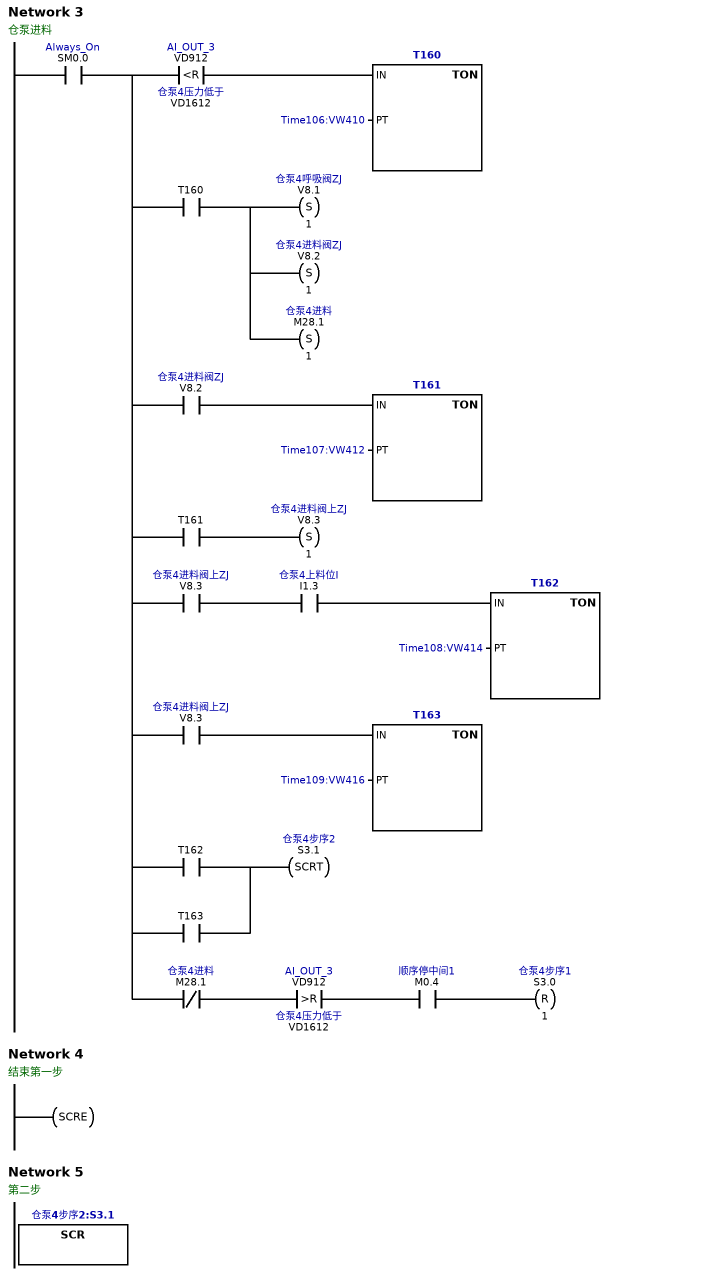
Network 3
// 仓泵进料
LD     Always_On:SM0.0
LPS
AR<    AI_OUT_3:VD912, 仓泵4压力低于:VD1612
TON    T160, Time106:VW410
LRD
A      T160
S      仓泵4呼吸阀ZJ:V8.1, 1
S      仓泵4进料阀ZJ:V8.2, 1
S      仓泵4进料:M28.1, 1
LRD
LPS
A      仓泵4进料阀ZJ:V8.2
TON    T161, Time107:VW412
LRD
A      T161
S      仓泵4进料阀上ZJ:V8.3, 1
LRD
A      仓泵4进料阀上ZJ:V8.3
A      仓泵4上料位I:I1.3
TON    T162, Time108:VW414
LPP
A      仓泵4进料阀上ZJ:V8.3
TON    T163, Time109:VW416
LRD
LD     T162
O      T163
ALD
SCRT   仓泵4步序2:S3.1
LPP
AN     仓泵4进料:M28.1
AR>    AI_OUT_3:VD912, 仓泵4压力低于:VD1612
A      顺序停中间1:M0.4
R      仓泵4步序1:S3.0, 1
Network 4
// 结束第一步
SCRE
Network 5
// 第二步 
LSCR   仓泵4步序2:S3.1
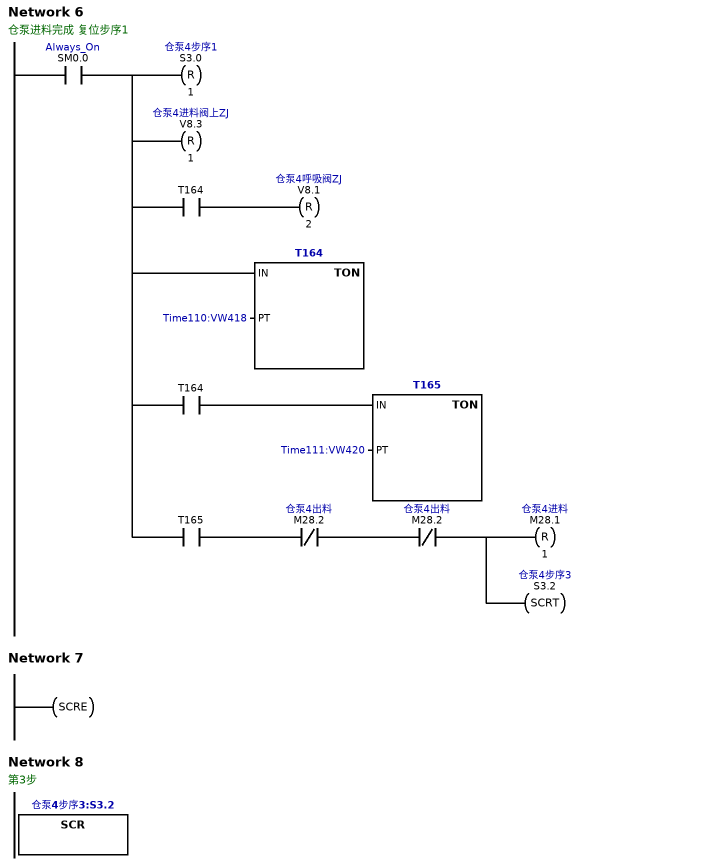
Network 6
// 仓泵进料完成 复位步序1
LD     Always_On:SM0.0
LPS
R      仓泵4步序1:S3.0, 1
R      仓泵4进料阀上ZJ:V8.3, 1
A      T164
R      仓泵4呼吸阀ZJ:V8.1, 2
LRD
TON    T164, Time110:VW418
LRD
A      T164
TON    T165, Time111:VW420
LPP
A      T165
AN     仓泵4出料:M28.2
AN     仓泵4出料:M28.2
R      仓泵4进料:M28.1, 1
SCRT   仓泵4步序3:S3.2
Network 7
SCRE
Network 8
// 第3步 
LSCR   仓泵4步序3:S3.2
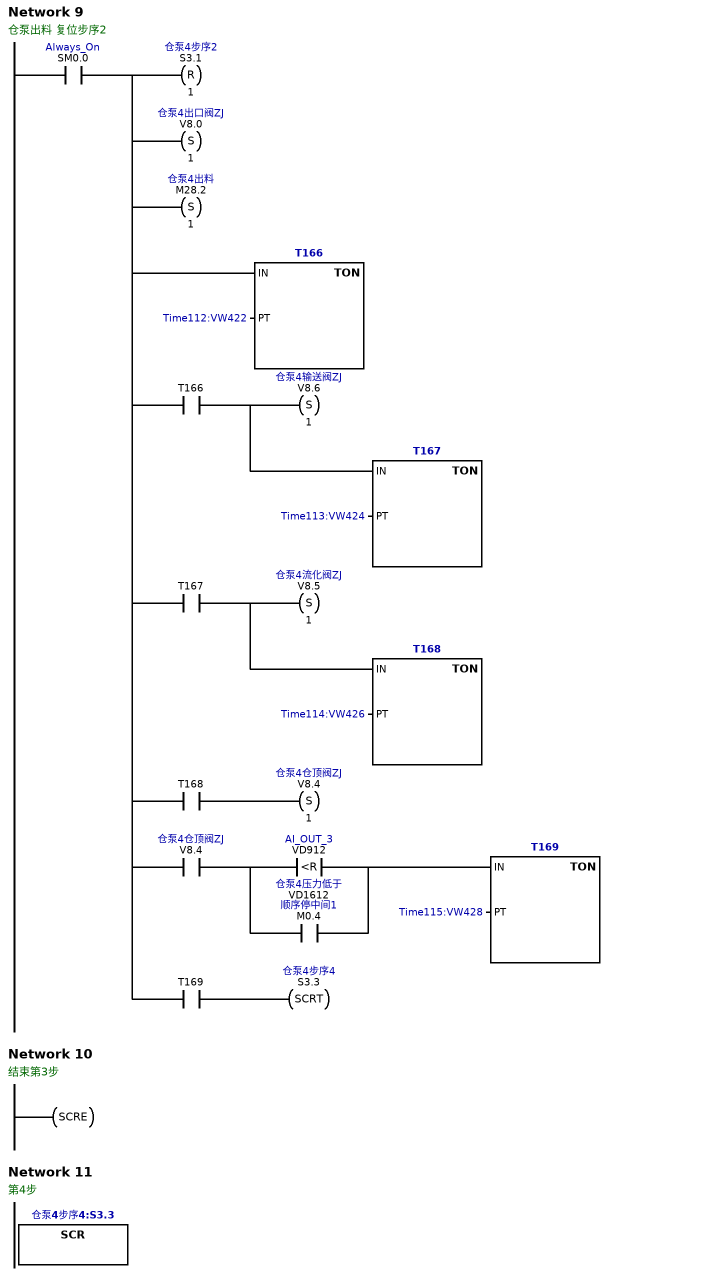
Network 9
// 仓泵出料 复位步序2
LD     Always_On:SM0.0
LPS
R      仓泵4步序2:S3.1, 1
S      仓泵4出口阀ZJ:V8.0, 1
S      仓泵4出料:M28.2, 1
TON    T166, Time112:VW422
A      T166
S      仓泵4输送阀ZJ:V8.6, 1
TON    T167, Time113:VW424
LRD
A      T167
S      仓泵4流化阀ZJ:V8.5, 1
TON    T168, Time114:VW426
LRD
A      T168
S      仓泵4仓顶阀ZJ:V8.4, 1
LRD
A      仓泵4仓顶阀ZJ:V8.4
LDR<   AI_OUT_3:VD912, 仓泵4压力低于:VD1612
O      顺序停中间1:M0.4
ALD
TON    T169, Time115:VW428
LPP
A      T169
SCRT   仓泵4步序4:S3.3
Network 10
// 结束第3步
SCRE
Network 11
// 第4步 
LSCR   仓泵4步序4:S3.3
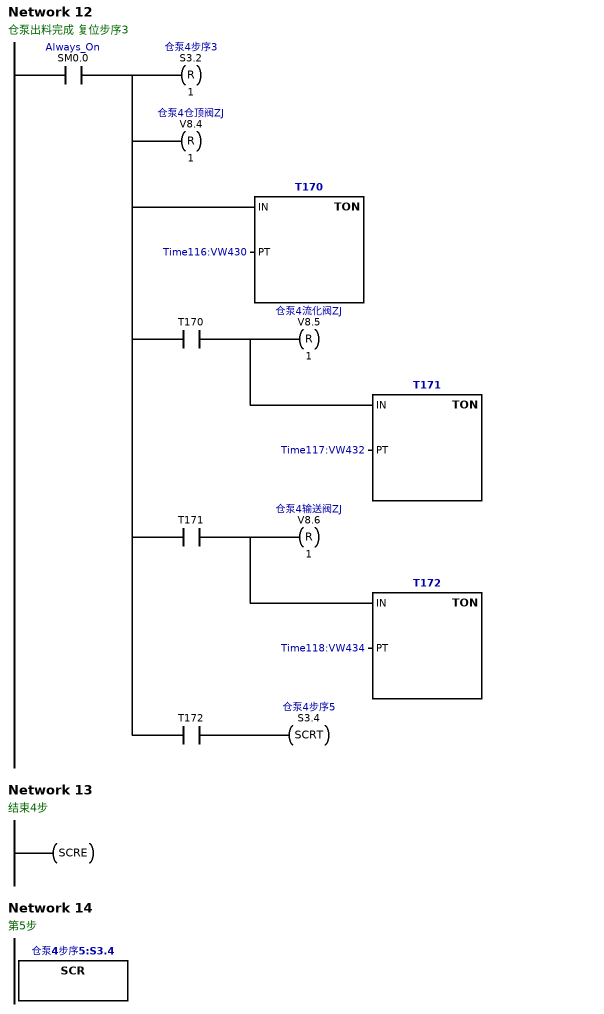
Network 12
// 仓泵出料完成 复位步序3
LD     Always_On:SM0.0
LPS
R      仓泵4步序3:S3.2, 1
R      仓泵4仓顶阀ZJ:V8.4, 1
TON    T170, Time116:VW430
A      T170
R      仓泵4流化阀ZJ:V8.5, 1
TON    T171, Time117:VW432
LRD
A      T171
R      仓泵4输送阀ZJ:V8.6, 1
TON    T172, Time118:VW434
LPP
A      T172
SCRT   仓泵4步序5:S3.4
Network 13
// 结束4步
SCRE
Network 14
// 第5步 
LSCR   仓泵4步序5:S3.4
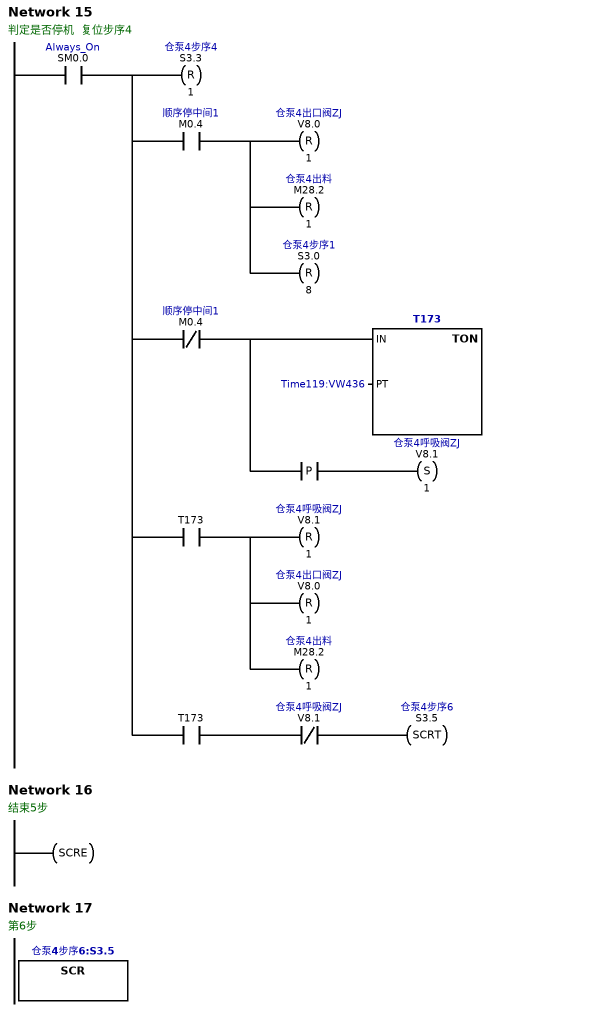
Network 15
// 判定是否停机  复位步序4 
LD     Always_On:SM0.0
LPS
R      仓泵4步序4:S3.3, 1
A      顺序停中间1:M0.4
R      仓泵4出口阀ZJ:V8.0, 1
R      仓泵4出料:M28.2, 1
R      仓泵4步序1:S3.0, 8
LRD
AN     顺序停中间1:M0.4
TON    T173, Time119:VW436
EU
S      仓泵4呼吸阀ZJ:V8.1, 1
LRD
A      T173
R      仓泵4呼吸阀ZJ:V8.1, 1
R      仓泵4出口阀ZJ:V8.0, 1
R      仓泵4出料:M28.2, 1
LPP
A      T173
AN     仓泵4呼吸阀ZJ:V8.1
SCRT   仓泵4步序6:S3.5
Network 16
// 结束5步
SCRE
Network 17
// 第6步 
LSCR   仓泵4步序6:S3.5
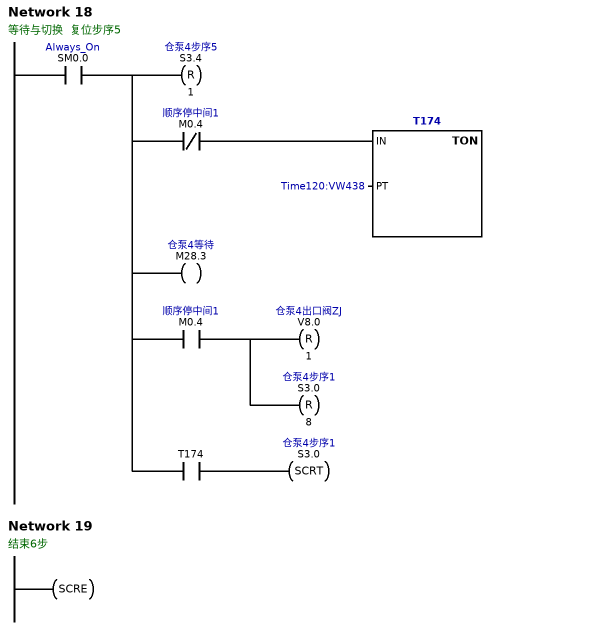
Network 18
// 等待与切换  复位步序5
LD     Always_On:SM0.0
LPS
R      仓泵4步序5:S3.4, 1
AN     顺序停中间1:M0.4
TON    T174, Time120:VW438
LRD
=      仓泵4等待:M28.3
LRD
A      顺序停中间1:M0.4
R      仓泵4出口阀ZJ:V8.0, 1
R      仓泵4步序1:S3.0, 8
LPP
A      T174
SCRT   仓泵4步序1:S3.0
Network 19
// 结束6步
SCRE
END_SUBROUTINE_BLOCK

SUBROUTINE_BLOCK 仓泵5:SBR24
TITLE=
VAR_OUTPUT
出口阀:BOOL;	// L0.0 
呼吸阀:BOOL;	// L0.1 
进料阀:BOOL;	// L0.2 
进料阀上:BOOL;	// L0.3 
仓顶阀:BOOL;	// L0.4 
流化阀:BOOL;	// L0.5 
输送阀:BOOL;	// L0.6 
END_VAR
BEGIN
